# EPICS substitutions: backup/mc1-rge1-test/tpmacApp/Db/motor.substitutions
file "db/motor.db"
{

# ADDR ---> axis #
# NOTE ---> 2 asyn ports: 1) lowel comms ("P0"), and 2) Motor Record ("motor")
pattern
{ P,             M,               MOTOR,   PORT,    ADDR, DESC,     DTYP }
{ "XF:23ID-Test", "{Dev-Ax:X}",	  "motor", "PO",    4,  "test axis 4 demo", asynMotor }
}
